Yaskawa INFORM job: R1_W13,15(0,0)KM-OKNEW.JBI

/JOB
//NAME R1_W13,15(0,0)KM-OKNEW
///FOLDERNAME SCIANA-NOWY-R2-KM
//POS
///NPOS 97,97,0,5,0,0
///TOOL 0
///POSTYPE PULSE
///PULSE
C00000=-147277,60026,-5631,-20277,85124,13806
C00001=-160074,80797,26825,-14512,73882,11454
C00002=-160843,86662,35984,-14314,71214,11522
C00003=-161140,89195,39907,-14253,70085,11558
C00004=-161775,90672,41778,-13960,69602,11398
C00005=-161140,89195,39907,-14253,70085,11558
C00006=-161063,90646,42469,-14364,69291,11681
C00007=-161063,90039,43321,-14440,68480,11781
C00008=-161063,90646,42469,-14364,69291,11681
C00009=-160899,91716,44118,-14490,68868,11791
C00010=-160588,94104,47162,-14712,68294,11972
C00011=-160899,91716,44118,-14490,68868,11791
C00012=-160602,89056,40019,-14540,70038,11748
C00013=-159834,82934,30508,-14714,72789,11666
C00014=-159775,78785,28717,-31049,45785,17949
C00015=-160744,86276,37714,-31059,43998,18135
C00016=-161118,89436,41574,-31127,43221,18241
C00017=-161766,90979,43527,-30761,42643,18122
C00018=-161118,89436,41574,-31127,43221,18241
C00019=-160989,91460,44001,-31494,42875,18446
C00020=-160696,93702,46857,-32104,42461,18773
C00021=-160989,91460,44001,-31494,42875,18446
C00022=-160955,90463,41510,-30968,43766,18115
C00023=-160955,91376,40496,-30399,44712,17757
C00024=-160955,90463,41510,-30968,43766,18115
C00025=-160580,87312,37646,-30905,44550,18008
C00026=-159608,79843,28641,-30904,46351,17821
C00027=-169578,72061,52050,-33550,65373,36771
C00028=-159639,102066,52849,-36627,118532,43382
C00029=-161230,98010,49947,-36645,117651,43000
C00030=-161874,96468,48906,-36639,117269,42855
C00031=-162414,97439,51471,-36313,116175,43029
C00032=-161874,96468,48906,-36639,117269,42855
C00033=-161681,87636,37192,-37728,115333,39463
C00034=-162202,89199,38314,-37765,115213,39280
C00035=-161681,87636,37192,-37728,115333,39463
C00036=-159221,89245,43122,-43634,115424,41269
C00037=-159607,86334,39462,-43925,115798,40898
C00038=-159221,89245,43122,-43634,115424,41269
C00039=-158510,90592,44026,-43670,115855,41410
C00040=-156755,94145,46551,-43727,116872,41780
C00041=-156215,89463,47666,-89737,91612,44965
C00042=-160258,86848,41994,-88867,88907,43909
C00043=-161076,86470,41042,-88663,88366,43712
C00044=-161752,88067,43044,-88493,87876,43890
C00045=-161076,86470,41042,-88663,88366,43712
C00046=-160594,87728,35116,-82489,91621,42752
C00047=-160965,85254,32003,-82415,91483,42439
C00048=-160594,87728,35116,-82489,91621,42752
C00049=-161203,99397,53897,-87809,93262,46482
C00050=-161203,99945,53017,-87887,93322,46099
C00051=-161203,99397,53897,-87809,93262,46482
C00052=-160420,100287,55440,-87942,93770,46729
C00053=-156570,105790,64558,-88393,96280,48111
C00054=-160137,66333,45297,-36257,70231,39255
C00055=-174783,98077,26040,-17019,52914,-20234
C00056=-174608,105356,36185,-17755,50551,-19749
C00057=-174540,108469,40544,-18090,49531,-19530
C00058=-174948,106579,37990,-17568,50029,-19783
C00059=-174535,106021,37238,-17896,50273,-19669
C00060=-174545,95141,46292,-21634,39727,-17290
C00061=-174613,91639,41667,-21115,40689,-17584
C00062=-174788,83471,31002,-20015,42870,-18217
C00063=-174723,64811,15244,-20023,42994,-18215
C00064=-174630,72581,24118,-20397,41940,-17819
C00065=-165301,85991,63683,-95469,38910,6878
C00066=-174940,70430,32149,-23153,35919,-16371
C00067=-174503,69857,31471,-23577,36151,-16189
C00068=-165282,98803,97625,-112321,41838,16779
C00069=-174585,69363,53194,-35008,24097,-10312
C00070=-172858,43893,24739,-32342,28495,-11698
C00071=-171579,71462,9368,-27845,35135,-13810
C00072=-159839,114570,69332,-85586,51587,5334
C00073=-162529,132656,93679,-89709,49247,8617
C00074=-162529,132656,93679,-89709,49247,8617
C00075=-174998,94453,36907,-27180,29568,-13493
C00076=-174582,93879,36167,-27626,29834,-13336
C00077=-152510,99797,82431,-97838,56868,14183
C00078=-172643,65899,17574,-22443,42662,-17134
C00079=-148864,54141,8521,-56122,89229,20941
C00080=-153335,95697,26029,-82409,110921,49707
C00081=-160363,104911,38709,-82349,112706,51438
C00082=-159280,86375,36579,-99137,101532,56181
C00083=-160497,97456,39712,-80225,111807,53659
C00084=-160755,98528,41110,-80015,111579,53795
C00085=-159089,75629,46556,-86176,101646,66755
C00086=-158598,89323,49372,-76132,110691,58792
C00087=-155696,101248,50108,-79244,114019,56233
C00088=-155378,96653,62951,-100962,108920,53706
C00089=-159710,92289,53440,-101347,105313,52189
C00090=-159988,90634,42470,-94412,106524,46277
C00091=-159803,91670,52086,-101491,105167,51947
C00092=-160062,92903,53649,-101325,105039,52119
C00093=-159968,90319,74690,-87370,106137,56061
C00094=-152319,115320,91112,-71043,111185,65415
C00095=-114526,45363,13216,-71043,111185,65415
C00096=-21612,48451,16538,1756,101829,65668
BC00000=327994,917845,549238
BC00001=327994,917845,549238
BC00002=327994,917845,549238
BC00003=327994,917845,549238
BC00004=327994,917845,549238
BC00005=327994,917845,549238
BC00006=327994,917845,549238
BC00007=327994,917845,549238
BC00008=327994,917845,549238
BC00009=327994,917845,549238
BC00010=327994,917845,549238
BC00011=327994,917845,549238
BC00012=327994,917845,549238
BC00013=327994,917845,549238
BC00014=352149,904506,798085
BC00015=352149,904506,798085
BC00016=352149,904506,798085
BC00017=352149,904506,798085
BC00018=352149,904506,798085
BC00019=352149,904506,798085
BC00020=352149,904506,798085
BC00021=352149,904506,798085
BC00022=352149,904506,798085
BC00023=352149,904506,798085
BC00024=352149,904506,798085
BC00025=352149,904506,798085
BC00026=352149,904506,798085
///LIMIT ON
BC00027=399927,939795,1076643
///LIMIT OFF
BC00028=313071,918337,578312
BC00029=313071,918337,578312
BC00030=313071,918337,578312
BC00031=313071,918337,578312
BC00032=313071,918337,578312
BC00033=313071,918337,578312
BC00034=313071,918337,578312
BC00035=313071,918337,578312
BC00036=313071,918337,578312
BC00037=313071,918337,578312
BC00038=313071,918337,578312
BC00039=313071,918337,578312
BC00040=313071,918337,578312
BC00041=361717,923326,729315
BC00042=361717,923326,729315
BC00043=361717,923326,729315
BC00044=361717,923326,729315
BC00045=361717,923326,729315
BC00046=361717,923326,729315
BC00047=361717,923326,729315
BC00048=361717,923326,729315
BC00049=361717,923326,729315
BC00050=361717,923326,729315
BC00051=361717,923326,729315
BC00052=361717,923326,729315
BC00053=361717,923326,729315
///LIMIT ON
BC00054=399927,926299,1076643
///LIMIT OFF
BC00055=390632,1409000,509189
BC00056=390632,1409000,509189
BC00057=390632,1409000,509189
BC00058=390632,1409000,509189
BC00059=390632,1409000,509189
BC00060=390632,1409000,509189
BC00061=390632,1409000,509189
BC00062=390632,1409000,509189
BC00063=380104,940780,622437
BC00064=380104,940781,622438
BC00065=380104,940781,622438
BC00066=380104,940781,622438
BC00067=380104,940781,622438
BC00068=380104,940781,524093
BC00069=380104,940781,622438
BC00070=380104,940781,622438
BC00071=391346,927863,633359
BC00072=391346,927863,633359
BC00073=391346,927863,633359
BC00074=391270,930791,636311
BC00075=391346,927863,633359
BC00076=391346,927863,633359
BC00077=346787,927863,633359
BC00078=391346,927863,633359
BC00079=355923,939638,739392
BC00080=332706,942259,475892
BC00081=332706,942259,475892
BC00082=332706,942259,475892
BC00083=332706,942259,475892
BC00084=332706,942259,475892
BC00085=332706,942258,475889
BC00086=332706,942259,475892
BC00087=332706,942259,475892
BC00088=333318,943748,720299
BC00089=333318,943748,720299
BC00090=333318,943748,720299
BC00091=333318,943748,720299
BC00092=333318,943748,720299
BC00093=333318,943748,720299
BC00094=333318,943748,720299
BC00095=335801,878385,876609
BC00096=132040,878385,876609
///POSTYPE BASE
///RECTAN
///RCONF 0,0,0,0,0,0,0,0,0,0,0,0,0,0,0,0,0,0,0,0,0,0,0,0
P00006=0.222,-3.123,-1.508,0.0000,0.0000,0.0000
P00021=-0.225,-6.128,-0.405,0.0000,0.0000,0.0000
P00022=0.222,-3.123,-1.508,0.0000,0.0000,0.0000
P00023=0.143,-0.036,0.682,0.0000,0.0000,0.0000
P00024=0.145,-0.552,1.326,0.0000,0.0000,0.0000
//INST
///DATE 2024/07/18 17:23
///ATTR SC,RW
///GROUP1 RB1,BS1
NOP
'r2_W13,15(0,0)
'
'Path S869
SFTOF
MOVJ C00000 BC00000 VJ=100.00
MOVJ C00001 BC00001 VJ=100.00
MOVL C00002 BC00002 V=100.0
MOVL C00003 BC00003 V=60.0
REFP 3 C00004 BC00004
CALL JOB:SEARCH-R1
SET P021 P006
SFTON P021
MOVL C00005 BC00005 V=60.0
MOVL C00006 BC00006 V=60.0
REFP 3 C00007 BC00007
CALL JOB:SEARCH-R1
SET P021 P006
SFTON P021
MOVL C00008 BC00008 V=60.0
MOVL C00009 BC00009 V=60.0
REFP 3 C00010 BC00010
CALL JOB:SEARCH-R1
SET P021 P006
SFTON P021
MOVL C00011 BC00011 V=60.0
MOVL C00012 BC00012 V=100.0
MOVL C00013 BC00013 V=333.3
'Path S870 (for W413)
SFTOF
MOVL C00014 BC00014 V=333.3
MOVL C00015 BC00015 V=200.0
MOVL C00016 BC00016 V=60.0
REFP 3 C00017 BC00017
CALL JOB:SEARCH-R1
SET P022 P006
SFTON P022
MOVL C00018 BC00018 V=60.0
MOVL C00019 BC00019 V=60.0
REFP 3 C00020 BC00020
CALL JOB:SEARCH-R1
SET P022 P006
SFTON P022
MOVL C00021 BC00021 V=60.0
MOVL C00022 BC00022 V=60.0
REFP 3 C00023 BC00023
CALL JOB:SEARCH-R1
SET P022 P006
SFTON P022
MOVL C00024 BC00024 V=60.0
MOVL C00025 BC00025 V=100.0
MOVL C00026 BC00026 V=100.0
COMM MOVJ C00027 BC00027 VJ=100.00
'Path S871 (for W414)
'ZLA KOLEJNOSC
SFTOF
MOVL C00028 BC00028 V=166.7
MOVL C00029 BC00029 V=166.7
MOVL C00030 BC00030 V=60.0
REFP 3 C00031 BC00031
CALL JOB:SEARCH-R1
SET P023 P006
SFTON P023
MOVL C00032 BC00032 V=60.0
MOVL C00033 BC00033 V=60.0
REFP 3 C00034 BC00034
CALL JOB:SEARCH-R1
SET P023 P006
SFTON P023
MOVL C00035 BC00035 V=60.0
MOVL C00036 BC00036 V=60.0
REFP 3 C00037 BC00037
CALL JOB:SEARCH-R1
SET P023 P006
SFTON P023
MOVL C00038 BC00038 V=60.0
MOVL C00039 BC00039 V=100.0
MOVL C00040 BC00040 V=100.0
'Path S872 (for W414)
SFTOF
MOVJ C00041 BC00041 VJ=100.00
MOVL C00042 BC00042 V=100.0
MOVL C00043 BC00043 V=60.0
REFP 3 C00044 BC00044
CALL JOB:SEARCH-R1
SET P024 P006
SFTON P024
MOVL C00045 BC00045 V=60.0
MOVL C00046 BC00046 V=60.0
REFP 3 C00047 BC00047
CALL JOB:SEARCH-R1
SET P024 P006
SFTON P024
MOVL C00048 BC00048 V=60.0
MOVL C00049 BC00049 V=60.0
REFP 3 C00050 BC00050
CALL JOB:SEARCH-R1
SET P024 P006
SFTON P024
MOVL C00051 BC00051 V=60.0
MOVL C00052 BC00052 V=100.0
MOVL C00053 BC00053 V=100.0
COMM MOVJ C00054 BC00054 VJ=100.00
COMM 'Path W873
COMM SFTOF
COMM SFTON P022
COMM MOVJ C00055 BC00055 VJ=100.00
COMM MOVL C00056 BC00056 V=400.0
COMM MOVL C00057 BC00057 V=100.0 PL=0
COMM REFP 1 C00058 BC00058
COMM REFP 2 C00059 BC00059
COMM MACRO1 MJ#(0) ARGF0
COMM ARCON
COMM SFTON P021
COMM MOVL C00060 BC00060 V=10.0
COMM ARCOF
COMM MOVL C00061 BC00061 V=400.0
COMM MOVL C00062 BC00062 V=1000.0
COMM SFTOF
'Path W916
SFTOF
SFTON P022
MOVJ C00063 BC00063 VJ=100.00
MOVL C00064 BC00064 V=100.0
MOVL C00065 BC00065 V=100.0 PL=0
REFP 1 C00066 BC00066
REFP 2 C00067 BC00067
MACRO1 MJ#(0) ARGF7
ARCON
SFTON P021
MOVL C00068 BC00068 V=12.5
ARCOF
MOVL C00069 BC00069 V=166.7
MOVL C00070 BC00070 V=250.0
SFTOF
'Path W917
SFTOF
SFTON P022
MOVJ C00071 BC00071 VJ=40.00
MOVL C00072 BC00072 V=250.0
MOVL C00073 BC00073 V=100.0 PL=0
MOVL C00074 BC00074 V=11.0
REFP 1 C00075 BC00075
REFP 2 C00076 BC00076
MACRO1 MJ#(0) ARGF7
ARCON
MOVL C00077 BC00077 V=12.5
ARCOF
MOVL C00078 BC00078 V=100.0
SFTOF
'Path VIA920
SFTOF
MOVJ C00079 BC00079 VJ=100.00
'Path W918
SFTOF
SFTON P024
MOVJ C00080 BC00080 VJ=100.00
MOVL C00081 BC00081 V=166.7
MOVL C00082 BC00082 V=100.0 PL=0
REFP 1 C00083 BC00083
REFP 2 C00084 BC00084
MACRO1 MJ#(0) ARGF10
ARCON
SFTON P023
MOVL C00085 BC00085 V=9.2
ARCOF
MOVL C00086 BC00086 V=166.7
MOVL C00087 BC00087 V=250.0
SFTOF
'Path W919
SFTOF
SFTON P024
MOVJ C00088 BC00088 VJ=100.00
MOVL C00089 BC00089 V=250.0
MOVL C00090 BC00090 V=100.0 PL=0
REFP 1 C00091 BC00091
REFP 2 C00092 BC00092
MACRO1 MJ#(0) ARGF10
ARCON
MOVL C00093 BC00093 V=9.2
SFTON P023
ARCOF
MOVL C00094 BC00094 V=100.0
MOVJ C00095 BC00095 VJ=100.00
SFTOF
MOVJ C00096 BC00096 VJ=100.00
END
